FUNCTION FC_5strConcatSeparator : T_DEFAULT_STR		// Concatenates 5 strings with given separator
VAR_INPUT
	iSeparator:		STRING := IING.STRING_UNDERSCORE;
	iStr1:			T_DEFAULT_STR;
	iStr2:			T_DEFAULT_STR;
	iStr3:			T_DEFAULT_STR;
	iStr4:			T_DEFAULT_STR;
	iStr5:			T_DEFAULT_STR;
END_VAR

FC_5strConcatSeparator := FC_2strConcatSeparator(iSeparator := iSeparator,
	iStr1 := FC_4strConcatSeparator(iSeparator := iSeparator, iStr1 := iStr1, iStr2 := iStr2, iStr3 := iStr3, iStr4 := iStr4), iStr2 := iStr5);

END_FUNCTION

(* stored: Version 1.1.0.1, ProductVersion 3.1.4026.18
   POU FC_5strConcatSeparator: Id {5a53e0ed-dbfb-4c88-88be-3959a12b21ed}, SpecialFunc None *)
